FUNCTION_BLOCK IndicateActivity EXTENDS ControlPrimitiveBase
VAR
	m_precondition: ValueExpression(EDataType.binary, TRUE, 0, '', TRUE);
// 	m_postcondition: ValueExpression(EDataType.binary, TRUE, 0, '', TRUE);
	m_postcondition: ComparisonExpression(EProcessVariables.LSC_RampEndWPCount, EComparisonType.greater, EDataType.numeric, FALSE, 0, '', TRUE);
	m_ptrIndic: POINTER TO ActivityIndicator;
	
	m_execTon: TON;
	m_blinkTon: TON;
END_VAR

SUPER^();

METHOD Abort : BOOL
VAR_INPUT
END_VAR
Abort := TRUE;
END_METHOD

(* Execution logic of this Control Primitive. *)
METHOD PROTECTED ExecuteInternal : BOOL
VAR_INPUT
	i_params	: Resi4MPM.ParameterSet;
END_VAR
VAR
	m_val: SNamedValue;
	m_dur: TIME;
END_VAR
m_val := i_params.Retrieve('duration_ms');
m_dur := LREAL_TO_TIME(m_val.Value.Numeric);

m_ptrIndic^.ResetDoneSignal();
ExecuteInternal := FALSE;
m_execTon(IN := TRUE, PT := m_dur);

IF m_execTon.Q THEN
	ExecuteInternal := TRUE;
	m_ptrIndic^.SetDoneSignal();
	m_execTon(IN := FALSE);
ELSE
	// "blink" the activity indicator
	m_blinkTon(IN := TRUE, PT := T#200MS);
	IF m_blinkTon.Q THEN
		m_ptrIndic^.FlipIndicator();
		m_blinkTon(IN := FALSE);
	END_IF
END_IF
END_METHOD

//FB_Init is always available implicitly and it is used primarily for initialization.
//The return value is not evaluated. For a specific influence, you can also declare the
//methods explicitly and provide additional code there with the standard initialization
//code. You can evaluate the return value.
METHOD FB_Init: BOOL
VAR_INPUT
    bInitRetains: BOOL; // TRUE: the retain variables are initialized (reset warm / reset cold)
    bInCopyCode: BOOL;  // TRUE: the instance will be copied to the copy code afterward (online change)
	
	i_id: UINT;
	i_ptrIndicator: POINTER TO ActivityIndicator;
END_VAR
m_id := i_id;
m_timeout := T#5S;
m_paramDefinition := 'duration_ms:UINT;';

Precondition := m_precondition;
Postcondition := m_postcondition;

m_ptrIndic := i_ptrIndicator;
END_METHOD

END_FUNCTION_BLOCK

(* stored: Version 1.1.0.1
   POU IndicateActivity: Id {5d1b302c-9c89-463d-8adf-0c8800c6d488}, SpecialFunc None
   Method Abort: Id {455eccc8-753f-4453-8457-a24b9976f13d}
   Method ExecuteInternal: Id {da7c07e4-7a02-41b2-8b16-3a55e97a34b5}
   Method FB_init: Id {21b1838c-cf3c-4a78-8fbb-bb36424196b1} *)
